// ---- POUs/Components/AxisDriver/Utilities/FB_AxisDistanceTrigger.TcPOU
FUNCTION_BLOCK FB_AxisDistanceTrigger
VAR_INPUT
	/// reset FB
	bReset				: BOOL;
	/// actual position
	fActualPos			: LREAL;
	/// trigger distance
	fTriggerDistance	: LREAL;
END_VAR
VAR_OUTPUT
	/// trigger output
	Q	: BOOL;
END_VAR
VAR PERSISTENT
	/// distance
	fDistance		: LREAL;
	/// actual ABS position
	fActualAbsPos	: LREAL;
	/// mirror ABS position
	fMirrorAbsPos	: LREAL;
	bInit			: BOOL;
END_VAR

fActualAbsPos := ABS(fActualPos);

IF bReset OR NOT bInit THEN
	bInit := TRUE;
	Q := FALSE;
	fMirrorAbsPos := fActualAbsPos;
	IF bReset THEN	
		fDistance := 0;
	END_IF

END_IF

IF fTriggerDistance <= 0 THEN
	Q := FALSE;
	RETURN;
END_IF

IF ABS(fActualAbsPos - fMirrorAbsPos) > fEpsilon THEN
	fDistance := fDistance + ABS(fActualAbsPos - fMirrorAbsPos);
	fMirrorAbsPos := fActualAbsPos;
END_IF

Q := fDistance >= fTriggerDistance;

END_FUNCTION_BLOCK

// ---- POUs/Components/AxisDriver/Utilities/FB_LimitSwitchRefSim.TcPOU
/// Axis driver limit switch
FUNCTION_BLOCK FB_LimitSwitchRefSim
VAR_INPUT
	/// Aktiviert die Logik
	bEnable					:BOOL;
	/// Position der Achse
	fPosition				:REAL;
	
	/// Endschalter (Oeffner)
	bLimitSwitch			:BOOL;
	/// Distanz Simuliertem Ref-Schalter zu Endschalter
	fRefLimitDistance		:REAL := 1.1;
	
	/// Referenzposition
	fRefPosition			:REAL;
	/// Pruefen des Positionsbereichs der Referenzposition
	fRefPosCheckArea		:REAL := 1;
END_VAR
VAR_OUTPUT
	/// Endschalter (Verzeogert)
	bLimitSwitchSim			:BOOL;
	/// Simulierter Ref Schalter
	bRefSwitchSim			:BOOL;
	
	/// Pruefung der Refpos OK
	bRefCheckOk				:BOOL;
END_VAR
VAR
	
END_VAR
VAR PERSISTENT
	fPosLatched			:REAL;
	bPosLatched			:BOOL;
END_VAR

(*
	Baustein um einen Ref-Schalter und Limitswitch mit 1 Eingang zu realisieren
	RE / 2015 / www.rmth.at
*)

// Limit muss hinter Ref liegen
IF (fRefLimitDistance <= fRefPosCheckArea) THEN
	fRefLimitDistance := fRefPosCheckArea + 0.1;
END_IF

IF NOT bEnable THEN
	bLimitSwitchSim := bLimitSwitch;
	bRefSwitchSim := bLimitSwitchSim;
	bRefCheckOk := FALSE;
	RETURN;
END_IF

// logik
IF bLimitSwitch THEN // (oeffner)
	fPosLatched := 0;
	bPosLatched := FALSE;	
	bLimitSwitchSim := TRUE; // limit ok
	bRefSwitchSim := FALSE; // kein referenz
	bRefCheckOk := FALSE;
	
ELSE
	// Position merken
	IF NOT bPosLatched THEN
		bPosLatched := TRUE;
		fPosLatched := fPosition;
	END_IF

	bRefSwitchSim := TRUE;
	bLimitSwitchSim := NOT (ABS(fPosition - fPosLatched) >= fRefLimitDistance);

	// Referenzpunkt pruefen
	bRefCheckOk := (ABS(fRefPosition - fPosLatched) <= fRefPosCheckArea) AND NOT bLimitSwitch;
END_IF

METHOD Reset : bool
VAR_INPUT
END_VAR
fPosLatched := 0;
bPosLatched := FALSE;
END_METHOD

END_FUNCTION_BLOCK

// ---- POUs/Components/AxisDriver/Utilities/F_SpeedReached.TcPOU
/// determines whether the actual speed (ABS value) is within the target-speed window
FUNCTION F_SpeedReached : BOOL
VAR_INPUT
	/// actual speed
	fActualSpeed: LREAL;
	/// target speed
	fTargetSpeed: LREAL;
	/// Override for axis and spindle
	fOverride: LREAL;
END_VAR

F_SpeedReached := F_SpeedWindowReached(fToleranceFactor:=0, fActualSpeed:=fActualSpeed, fTargetSpeed:=fTargetSpeed, fOverride:=fOverride);

END_FUNCTION

// ---- POUs/Components/AxisDriver/Utilities/F_SpeedWindowReached.TcPOU
/// determines whether the actual speed (ABS value) is within the target-speed window
FUNCTION F_SpeedWindowReached : BOOL
VAR_INPUT
	/// factor for tolerance (default: 0.1)
	fToleranceFactor: REAL;
	/// actual speed
	fActualSpeed: LREAL;
	/// target speed
	fTargetSpeed: LREAL;
	/// Override for axis and spindle
	fOverride: LREAL;
END_VAR
VAR CONSTANT
	fDefaultfToleranceFactor: REAL := 0.1;
END_VAR
VAR
	fTol: LREAL;
	fMin: LREAL;
	fMax: LREAL;
	fAct: LREAL;
	fTar: LREAL;
END_VAR

// validate tolerance factor
IF fToleranceFactor <= 0 THEN
	fToleranceFactor:=fDefaultfToleranceFactor;
END_IF

// calc tolerance window and ABS values
fTar:=fTargetSpeed*(fOverride/100);
fTol:=ABS(fTar) * fToleranceFactor;
fMin:=ABS(fTar) - fTol;
fMax:=ABS(fTar) + fTol;
fAct:=ABS(fActualSpeed);

F_SpeedWindowReached := fAct >= fMin AND fAct <= fMax;

END_FUNCTION

// ---- POUs/Components/AxisDriver/Utilities/F_TargetReached.TcPOU
FUNCTION F_TargetReached : BOOL
VAR_INPUT
	fCurrentPos: LREAL;
	fTargetPos: LREAL;
END_VAR

F_TargetReached := F_TargetWindowReached(fCurrentPos, fTargetPos, fEpsilon);

END_FUNCTION

// ---- POUs/Components/AxisDriver/Utilities/F_TargetReachedOrHigher.TcPOU
FUNCTION F_TargetReachedOrHigher : BOOL
VAR_INPUT
	fCurrentPos: LREAL;
	fTargetPos: LREAL;
END_VAR


F_TargetReachedOrHigher := fCurrentPos >= (fTargetPos - fEpsilon);

END_FUNCTION

// ---- POUs/Components/AxisDriver/Utilities/F_TargetReachedOrLower.TcPOU
FUNCTION F_TargetReachedOrLower : BOOL
VAR_INPUT
	fCurrentPos: LREAL;
	fTargetPos: LREAL;
END_VAR


F_TargetReachedOrLower := fCurrentPos <= (fTargetPos + fEpsilon);

END_FUNCTION

// ---- POUs/Components/CylinderDriver/FB_Cylinder_Ui.TcPOU
FUNCTION_BLOCK PUBLIC FB_Cylinder_Ui EXTENDS FB_ManualUiBase
VAR_INPUT
	// Handbetrieb nach GRST
	bManual_HP				: BOOL;
	/// Handbetrieb nach AST
	bManual_WP				: BOOL;
	// Enable Mp
	bEnable_Mp				: BOOL;
END_VAR
VAR_IN_OUT
	// cylinder reference
	fbCylinder				: FB_CylinderEx;
	// hmi control IN
	stHMIControlIn			: ST_HMI_MANUAL_CYLINDER_IN;
	// hmi control IN
	stHMIControlOut			: ST_HMI_MANUAL_CYLINDER_OUT;	
END_VAR
VAR_OUTPUT
	diColorSelectedItem: UDINT;
	/// 0=Undefiniert
	/// 1=Fehler
	/// 2=In GRST (eingefahren)
	/// 3=In AST (ausgefahren) 
	iState: INT;
	diColorState	: UDINT;
	sState			: STRING;
	stState			: ST_Text;
END_VAR

stName.wsName := TO_WSTRING(fbCylinder.sName);
fbCylinder.diObjectIndex := diObjectIndex;
fbCylinder.diSelectedObjectIndex := diSelectedObjectIndex;
fbCylinder.bEnableManual := bEnableManual;
fbCylinder.bManual_HP := stHMIControlIn.stButtonHp.bClick OR ((diObjectIndex = diSelectedObjectIndex) AND stHMIControlIn.stButtonHp.bClick) ;
fbCylinder.bManual_WP := stHMIControlIn.stButtonWp.bClick OR ((diObjectIndex = diSelectedObjectIndex) AND stHMIControlIn.stButtonWp.bClick);

IF ((diObjectIndex = diSelectedObjectIndex) AND stHMIControlIn.stButtonMp.bClick) AND ((fbCylinder.eValveType = E_ValveType.eValvetype_5_3_lock) OR (fbCylinder.eValveType = E_ValveType.eValvetype_5_3_unlock)) THEN
	fbCylinder.ClearOuts();
END_IF

IF (diObjectIndex = diSelectedObjectIndex)AND (diObjectIndex <> 0) AND bEnableManual  THEN
	bManualActive := TRUE;
	stHMIControlOut.bVisible := TRUE;
	stHMIControlOut.stButtonHp.stName := CONST.stTextListGlobal.stText_Hp;
	stHMIControlOut.stButtonMp.stName := CONST.stTextListGlobal.stText_Mp;
	stHMIControlOut.stButtonWp.stName := CONST.stTextListGlobal.stText_Wp;
	stHMIControlOut.stObjectName.wsName := stHMIControlOut.stObjectName.wsNameId := TO_WSTRING(fbCylinder.sName);
	stHMIControlOut.stButtonHp.stColor.color := F_ColorToStringHexColor(STATICS.stColor.Theme);
	stHMIControlOut.stButtonWp.stColor.color := F_ColorToStringHexColor(STATICS.stColor.Theme);
	stHMIControlOut.bMpVisible := bEnable_Mp;
	stHMIControlOut.stButtonMp.stColor.color := F_ColorToStringHexColor(STATICS.stColor.Theme);	
	
	IF fbCylinder.bIn_HP THEN
		stHMIControlOut.stButtonHp.stColor.color := F_ColorToStringHexColor(STATICS.stColor.LimeGreen);
	ELSIF fbCylinder.bIn_WP THEN
		stHMIControlOut.stButtonWp.stColor.color := F_ColorToStringHexColor(STATICS.stColor.LimeGreen);
	END_IF
ELSIF bManualActive THEN
	bManualActive := FALSE;
	stHMIControlOut.bVisible := FALSE;
END_IF

iState := fbCylinder.iStatus;

CASE iState OF 
	1:
		sState:=fbCylinder.sErrText;
		diColorState:= STATICS.stColor.Red;
		stState.wsName := "error";
		stState.wsNameId := "error";
		stState.nNameId := 1;
	2:
		sState:= F_GetTranslatedTxtLib('Zylinder in HP', eLanguage);
		diColorState:= STATICS.stColor.Green;
		stState.wsName := "hp";
		stState.wsNameId := "inhomepos";
		stState.nNameId := 2;		
	3:
		sState:=F_GetTranslatedTxtLib('Zylinder in WP', eLanguage);
		diColorState:= STATICS.stColor.Green;
		stState.wsName := "wp";
		stState.wsNameId := "wp";
		stState.nNameId := 3;
ELSE
	sState:=F_GetTranslatedTxtLib(' Undefiniert ' , eLanguage);	
	diColorState:= STATICS.stColor.Orange;
	stState.wsName := "undifined";
	stState.wsNameId := "undifined";
	stState.nNameId := 0;	
END_CASE


IF (diObjectIndex=diSelectedObjectIndex) THEN
	diColorSelectedItem:=STATICS.stColor.LimeGreen;
ELSE
	diColorSelectedItem:=STATICS.stColor.Gray;	
END_IF

A_StateMapping();

ACTION A_StateMapping:
IF NOT __ISVALIDREF(stStateObject) THEN
	RETURN;
END_IF

// state mapping
stStateObject.stState := stState;
stStateObject.nIndexColor := diColorSelectedItem;
//stStateObject.stValue.wsName := "HP/WP";
END_ACTION

METHOD Control_Hp : BOOL
IF bEnableManual THEN
	bManual_HP:=TRUE;
END_IF
END_METHOD

METHOD Control_Wp : BOOL
IF bEnableManual THEN
	bManual_WP:=TRUE;
END_IF
END_METHOD

END_FUNCTION_BLOCK

// ---- POUs/Components/DriveFu/FB_Drive.TcPOU
FUNCTION_BLOCK FB_Drive
VAR_IN_OUT
	bInHome: BOOL;
END_VAR
VAR_INPUT
	/// component active flag
	bActive: BOOL;
	/// Objekt Name (BMK)
	stName				:ST_Text;
	/// Sicherheit = Freigabe von Bewegungen
	bSafetyOk			:BOOL;
	/// Motorschutz OK
	bMotorprotectionOk		:BOOL;

	// Hand
	///Objekt Index
	diObjectIndex: DINT;
	///Ausgewähltes Objekt in der Visu
	diSelectedObjectIndex	:DINT;
	/// Gibt den Handbetrieb frei
	bEnableManual: BOOL;
	// Handbetrieb nach GRST
	bManual_Reverse: BOOL;
	/// Handbetrieb nach AST
	bManual_Forward: BOOL;
	///	 Handbetrieb Stop
	bManual_Stop :BOOL;
	//	Type Handbetrieb
	// 1 = Tippen
	// 2 = Speichern
	iType : INT;
	
	///	Zus. Freigabe für HP Ausgang schalten	
	bFreigabe_Reverse: BOOL := TRUE;
	///	Zus. Freigabe für WP Ausgang schalten	
	bFreigabe_Forward: BOOL := TRUE;
END_VAR
VAR_OUTPUT	
	/// Summenfehler
	bError		:BOOL;
	/// Fehlerinformation
	sErrText	:ST_Text;
	/// 0=Undefiniert
	/// 1=Fehler
	/// 2=Stillstand OK
	/// 3=Vorwärts
	///	4=Rückwärts 
	iStatus: INT;	

	bInit_OK: BOOL;
	
	bDrive_Reverse_Out: BOOL;
	bDrive_Forward_Out: BOOL;
END_VAR
VAR
	iTypeOld : INT;
	tofForward: TOF;
	tofReverse: TOF;
	
	bDrive_Reverse: BOOL;
	bDrive_Forward: BOOL;
END_VAR

(*FB Drive für Antriebe*)
(*Erstellt von Stephan Schöchtner RMTH GmbH*)
(*21.März.2018*)

tofForward();
tofForward.IN := bManual_Forward;

tofReverse();
tofReverse.IN := bManual_Reverse;


// Initialisierung
IF NOT bInit_OK THEN
	M_Init();	
	bInit_OK :=TRUE;
END_IF

sERRText := CONST.stTextListGlobal.stText_notext;

//Fehler
bError := FALSE;
IF NOT bMotorprotectionOK THEN
	bError := TRUE;
	sErrText := F_CreateDynText("Motorschutz", 0);
END_IF

// Bei Typumschaltung im laufenden Betrieb STOP
IF iType <> iTypeOld THEN
	iTypeOld := iType;
	M_Stop();
END_IF

IF (diObjectIndex = diSelectedObjectIndex) THEN
	// Tippen mit Wendeschützumschaltung und Typumschaltung
	CASE iType OF	//Tippen
	
		1:
			IF bManual_Forward AND NOT bManual_Stop THEN
				bDrive_Reverse := FALSE;
				IF NOT tofReverse.Q THEN
					M_Start_Forward();
				END_IF
			ELSIF bManual_Reverse AND NOT bManual_Stop THEN
				bDrive_Forward := FALSE;
				IF NOT tofForward.Q THEN
					M_Start_Reverse();
				END_IF
			ELSE
				M_Stop();
				//M_Start_Forward := FALSE;
				//M_Start_Reverse := FALSE;
			END_IF
		2:						//Speichern
			IF bManual_Forward AND NOT bManual_Stop THEN
				bDrive_Reverse := FALSE;
				IF NOT tofReverse.Q THEN
					M_Start_Forward();
				END_IF
			ELSIF bManual_Reverse AND NOT bManual_Stop THEN
				bDrive_Forward := FALSE;
				IF NOT tofForward.Q THEN
					M_Start_Reverse();
				END_IF
			END_IF
			IF bManual_Stop THEN
				M_Stop();
				//M_Start_Forward := FALSE;
				//M_Start_Reverse := FALSE;
			END_IF	
	ELSE
		//no type selected
		bError := TRUE;
		sErrText := F_CreateDynText("Handbetriebstyp falsch", 0);
		M_Stop();
	END_CASE
END_IF

IF bError THEN
	istatus := 1;
ELSIF NOT bDrive_Forward AND NOT bDrive_Reverse THEN
	iStatus := 2;
ELSIF bDrive_Forward THEN
	iStatus := 3;
ELSIF bDrive_Reverse THEN
	iStatus := 4;
END_IF


bDrive_Reverse_Out:= bDrive_Reverse AND bFreigabe_Reverse AND bSafetyOk AND bMotorprotectionOk;
bDrive_Forward_Out:= bDrive_Forward AND bFreigabe_Forward AND bSafetyOk AND bMotorprotectionOk;

IF NOT bSafetyOk THEN
	bDrive_Reverse:=FALSE;
	bDrive_Reverse_Out:=FALSE;

	bDrive_Forward:=FALSE;
	bDrive_Forward_Out:=FALSE;	
END_IF


//Wegfahrsperre
IF bError THEN
	M_Stop();
END_IF

METHOD M_Init : BOOL
VAR_INPUT
END_VAR
bDrive_Forward := FALSE;
bDrive_Reverse := FALSE;
tofForward.IN := FALSE;
tofForward.PT := T#150MS;
tofReverse.IN := FALSE;
tofReverse.PT := T#150MS;
END_METHOD

METHOD M_Reset : BOOL
VAR_INPUT
END_VAR
END_METHOD

METHOD M_Start_Forward : BOOL
VAR_INPUT
END_VAR
bDrive_Reverse := FALSE;
bDrive_Forward := TRUE;
END_METHOD

METHOD M_Start_Reverse : BOOL
VAR_INPUT
END_VAR
bDrive_Reverse := TRUE;
bDrive_Forward := FALSE;
END_METHOD

METHOD M_Stop : BOOL
VAR_INPUT
END_VAR
	bDrive_Reverse := FALSE;
	bDrive_Forward := FALSE;
END_METHOD

END_FUNCTION_BLOCK

// ---- POUs/Components/DriveFu/FB_Drive_Ui.TcPOU
FUNCTION_BLOCK PUBLIC FB_Drive_Ui EXTENDS FB_ManualUiBase
VAR_INPUT
	// Handbetrieb Rückwärts
	bManual_Reverse				: BOOL;
	/// Handbetrieb Vorwärts
	bManual_Forward				: BOOL;
	//	Stop
	bManual_Stop				: BOOL;
	//	Type Handmodus
		// 1 = Tippen
		// 2 = Speichern
	iType						: INT;
END_VAR
VAR_IN_OUT
	// drive reference
	fbDrive				: FB_Drive;
	// hmi control IN
	stHMIControlIn			: ST_HMI_MANUAL_DRIVE_IN;
	// hmi control OUT
	stHMIControlOut			: ST_HMI_MANUAL_DRIVE_OUT;	
END_VAR
VAR_OUTPUT
	diColorSelectedItem: UDINT;
	/// 0=Undefiniert
	/// 1=Fehler
	iState: INT;
	diColorState	: UDINT;
	sState			: STRING;
	stState			: ST_Text;
END_VAR

stName := fbDrive.stName;

fbDrive.diObjectIndex := diObjectIndex;
fbDrive.diSelectedObjectIndex := diSelectedObjectIndex;
fbDrive.bEnableManual := bEnableManual;
//fbDrive.bManual_Reverse := bManual_Reverse;
//fbDrive.bManual_Forward := bManual_Forward;
//fbDrive.bManual_Stop := bManual_Stop;
fbDrive.iType := iType;

IF (diSelectedObjectIndex = diObjectIndex)AND (diObjectIndex <> 0) AND bEnableManual THEN
	bManualActive := TRUE;
	stHMIControlOut.bVisible := TRUE;
	stHMIControlOut.stObjectName := fbDrive.stName;
	stHMIControlOut.stButtonJogPos.stName := CONST.stTextListGlobal.stText_Positive;
	stHMIControlOut.stButtonJogNeg.stName := CONST.stTextListGlobal.stText_Negative;
	stHMIControlOut.stButtonStop.stName := CONST.stTextListGlobal.stText_Stop;
	stHMIControlOut.aDriveModeName[0] :=  CONST.stTextListGlobal.stText_Mode_StartStop;
	stHMIControlOut.aDriveModeName[1] :=  CONST.stTextListGlobal.stText_Mode_Jog;
	
	CASE stHMIControlIn.eJogMode OF
		
	E_Drive_JogMode.eJogMode_0 :
			IF stHMIControlIn.stButtonStop.bClick THEN
				fbDrive.M_Stop();
			ELSIF stHMIControlIn.stButtonJogPos.bClick THEN
				fbDrive.M_Start_Forward();
			ELSIF stHMIControlIn.stButtonJogNeg.bClick THEN	
				fbDrive.M_Start_Reverse();	
			END_IF
	E_Drive_JogMode.eJogMode_1 :
		IF stHMIControlIn.stButtonJogPos.bClick THEN
			fbDrive.M_Start_Forward();
		ELSIF stHMIControlIn.stButtonJogNeg.bClick THEN	
			fbDrive.M_Start_Reverse();	
		ELSE
			fbDrive.M_Stop();	
		END_IF				
	END_CASE
	stHMIControlOut.stButtonJogPos.stColor.color := F_ColorToStringHexColor(STATICS.stColor.Theme);
	stHMIControlOut.stButtonJogNeg.stColor.color := F_ColorToStringHexColor(STATICS.stColor.Theme);
	stHMIControlOut.stButtonStop.stColor.color := F_ColorToStringHexColor(STATICS.stColor.Red);
	IF fbDrive.bDrive_Forward_Out THEN
		stHMIControlOut.stButtonJogPos.stColor.color := F_ColorToStringHexColor(STATICS.stColor.LimeGreen);	
	END_IF
	IF fbDrive.bDrive_Reverse_Out THEN
		stHMIControlOut.stButtonJogNeg.stColor.color := F_ColorToStringHexColor(STATICS.stColor.LimeGreen);	
	END_IF	
	
	stHMIControlOut.stState	:= stState;	
ELSIF bManualActive THEN
	bManualActive := FALSE;
	stHMIControlOut.bVisible := FALSE;
END_IF

iState := fbDrive.iStatus;

CASE iState OF 
	1:
		sState:= TO_STRING( fbDrive.sErrText.wsName );
		diColorState:= STATICS.stColor.Red;
		stState.wsName := "error";
		stState.wsNameId := "error";
		stState.nNameId := 1;
	2:
		sState:= ('Stillstand OK');
		diColorState:= STATICS.stColor.Gray;
		stState.wsName := "notmoveing";
		stState.wsNameId := "notmoveing";
		stState.nNameId := 2;
	3:
		sState:= ('Betrieb Vorwärts');
		diColorState:= STATICS.stColor.Green;
		stState.wsName := "movepositive";
		stState.wsNameId := "movepositive";
		stState.nNameId := 3;
	4:
		sState:= ('Betrieb Rückwärts');
		diColorState:= STATICS.stColor.Green;
		stState.wsName := "movenegative";
		stState.wsNameId := "movenegative";
		stState.nNameId := 4;		
				
ELSE
	sState:= (' Undefiniert ');	
	diColorState:= STATICS.stColor.Orange;	
	stState.wsName := "undifined";
	stState.wsNameId := "undifined";
	stState.nNameId := 0;
END_CASE


IF (diObjectIndex=diSelectedObjectIndex) THEN
	diColorSelectedItem:=STATICS.stColor.LimeGreen;
ELSE
	diColorSelectedItem:=STATICS.stColor.Gray;	
END_IF

A_StateMapping();

ACTION A_StateMapping:
IF NOT __ISVALIDREF(stStateObject) THEN
	RETURN;
END_IF

// state mapping
stStateObject.stState := stState;
stStateObject.nIndexColor := diColorSelectedItem;
//stStateObject.stValue.wsName := "mov/stp";
END_ACTION

METHOD Control_Start_Forward : BOOL
IF bEnableManual THEN
	fbDrive.bManual_Reverse := FALSE;
	fbDrive.bManual_Forward := TRUE;
	fbDrive.bManual_Stop := FALSE;	
END_IF
END_METHOD

METHOD Control_Start_Reverse : BOOL
IF bEnableManual THEN
	fbDrive.bManual_Reverse := TRUE;
	fbDrive.bManual_Forward := FALSE;
	fbDrive.bManual_Stop := FALSE;	
END_IF
END_METHOD

METHOD Control_Stop : BOOL
IF bEnableManual THEN
	fbDrive.bManual_Reverse := FALSE;
	fbDrive.bManual_Forward := FALSE;
	fbDrive.bManual_Stop := TRUE;	
END_If
END_METHOD

END_FUNCTION_BLOCK

// ---- POUs/Components/DriveFu/FB_DriveFuAx_Ui.TcPOU
FUNCTION_BLOCK PUBLIC FB_DriveFuAx_Ui EXTENDS FB_ManualUiBase
VAR_INPUT
	// velocity
	fVelocity				: REAL := 1;	
	// additional enable flag for pos. direction
	bEnablePos				: BOOL := TRUE;
	// additional enable flag for neg. direction
	bEnableNeg				: BOOL := TRUE;	
	// manual jog neg.
	bJobN					: BOOL;
	// manual jog pos.
	bJogP					: BOOL;
	// manual stop
	bStop					: BOOL;
END_VAR
VAR_IN_OUT
	// axis reference
	fbAxis				: FB_AxisDriver;
	// hmi control IN
	stHMIControlIn		: ST_HMI_MANUAL_DRIVE_IN;
	// hmi control OUT
	stHMIControlOut		: ST_HMI_MANUAL_DRIVE_OUT;
END_VAR
VAR_OUTPUT	
	diColorSelectedItem: UDINT;
	/// 0=undefined 
	/// 1=error
	/// 2=moving pos. 
	/// 3=moving neg.
	/// 4=standstill
	/// 5=in sync
	iState			: INT;
	diColorState	: UDINT;
	sState			: STRING;
	stState			: ST_Text;
END_VAR
VAR
	stAxisState		: Tc2_MC2.ST_AxisStatus;
END_VAR

// AX5000 UI like frequency inverter (FU)

stName := fbAxis.Name;

// inactive -> reset & exit
IF NOT fbAxis.Active THEN
	stState := CONST.stTextListGlobal.stText_notext;
	iState := 0;// 0=undefined
	A_StateMapping();
	RETURN;
END_IF

IF (diSelectedObjectIndex = diObjectIndex)AND (diObjectIndex <> 0) AND bEnableManual THEN
	bManualActive := TRUE;
	stHMIControlOut.bVisible := TRUE;
	stHMIControlOut.stObjectName := fbAxis.Name;
	stHMIControlOut.stButtonJogPos.stName := CONST.stTextListGlobal.stText_Positive;
	stHMIControlOut.stButtonJogNeg.stName := CONST.stTextListGlobal.stText_Negative;
	stHMIControlOut.stButtonStop.stName := CONST.stTextListGlobal.stText_Stop;
	stHMIControlOut.aDriveModeName[0] :=  CONST.stTextListGlobal.stText_Mode_StartStop;
	stHMIControlOut.aDriveModeName[1] :=  CONST.stTextListGlobal.stText_Mode_Jog;
	
	CASE stHMIControlIn.eJogMode OF
		
	E_Drive_JogMode.eJogMode_0 :
			IF stHMIControlIn.stButtonStop.bClick THEN
				fbAxis.Stop();
			ELSIF stHMIControlIn.stButtonJogPos.bClick THEN
				fbAxis.MoveVel(fVelocity, MC_Direction.MC_Positive_Direction);
			ELSIF stHMIControlIn.stButtonJogNeg.bClick THEN	
				fbAxis.MoveVel(fVelocity, MC_Direction.MC_Negative_Direction);	
			END_IF
	E_Drive_JogMode.eJogMode_1 :
		fbAxis.JogExVel(((bJobN OR stHMIControlIn.stButtonJogNeg.bClick) AND bEnableNeg),
						((bJogP OR stHMIControlIn.stButtonJogPos.bClick) AND bEnablePos),
						fVelocity, E_JogMode.MC_JOGMODE_CONTINOUS);			
	END_CASE
	stHMIControlOut.stButtonJogPos.stColor.color := F_ColorToStringHexColor(STATICS.stColor.Theme);
	stHMIControlOut.stButtonJogNeg.stColor.color := F_ColorToStringHexColor(STATICS.stColor.Theme);
	stHMIControlOut.stButtonStop.stColor.color := F_ColorToStringHexColor(STATICS.stColor.Red);
	IF iState = 2 THEN // 2 = moving neg
		stHMIControlOut.stButtonJogPos.stColor.color := F_ColorToStringHexColor(STATICS.stColor.LimeGreen);	
	END_IF
	IF iState = 3 THEN // 3 = moving neg
		stHMIControlOut.stButtonJogNeg.stColor.color := F_ColorToStringHexColor(STATICS.stColor.LimeGreen);	
	END_IF	
	
	stHMIControlOut.stState	:= stState;	
ELSIF bManualActive THEN
	bManualActive := FALSE;
	stHMIControlOut.bVisible := FALSE;
END_IF

A_StateMapping();

ACTION A_StateMapping:
IF (diObjectIndex = diSelectedObjectIndex) THEN
	diColorSelectedItem := STATICS.stColor.LimeGreen;
ELSE
	diColorSelectedItem := STATICS.stColor.Gray;	
END_IF

bError := fbAxis.State = E_ComponentState.eComponentState_error;
IF bError THEN
	stErrorText := F_CreateDynText(fbAxis.ClearText, 0);
ELSE
	stErrorText := CONST.stTextListGlobal.stText_notext;
END_IF

// Status
stAxisState := fbAxis.AxisState;
IF bError THEN
	iState := 1; // 1=Fehler; 
	diColorState:= STATICS.stColor.Red;
	stState.wsNameId := "error";
	stState.wsName := "error";
	stState.nNameId :=1;
ELSIF stAxisState.Moving AND stAxisState.PositiveDirection THEN
	iState := 2; // 2=Fahrt Positiv; 
	diColorState:= STATICS.stColor.Green;
	stState.wsNameId := "movepositive";
	stState.wsName := "movepositive";
	stState.nNameId :=2;
ELSIF stAxisState.Moving AND stAxisState.NegativeDirection THEN
	iState := 3; // 3=Fahrt Negativ;
	diColorState:= STATICS.stColor.Green;
	stState.wsNameId := "movenegative";
	stState.wsName := "movenegative";
	stState.nNameId :=3;
ELSIF stAxisState.Coupled THEN
	iState := 5; // 5=Synchron
	diColorState:= STATICS.stColor.LightSkyBlue;
	stState.wsNameId := "coupled";
	stState.wsName := "coupled";
	stState.nNameId :=5;
ELSIF NOT stAxisState.Moving THEN
	iState := 4; // 4=Stillstand
	diColorState:= STATICS.stColor.Gray;
	stState.wsNameId := "notmoveing";
	stState.wsName := "notmoveing";
	stState.nNameId :=4;
ELSE
	iState := 0;// 0=Undefiniert
	diColorState:= STATICS.stColor.Orange;
	stState.wsNameId := "undifined";
	stState.wsName := "undifined";
	stState.nNameId :=0;
END_IF

IF NOT __ISVALIDREF(stStateObject) THEN
	RETURN;
END_IF

// state mapping
stStateObject.stState := stState;
stStateObject.nIndexColor := diColorSelectedItem;
//stStateObject.stValue.wsName := "mov/stp";
END_ACTION

END_FUNCTION_BLOCK

// ---- POUs/HMI/Utilities/F_AlarmPrioToText.TcPOU
FUNCTION F_AlarmPrioToText : ST_Text
VAR_INPUT
	ePriority : E_AlarmPriority;
END_VAR

			
CASE ePriority OF
	E_AlarmPriority.Error:
		F_AlarmPrioToText := Const.stTextListGlobal.stText_Error;
		
	E_AlarmPriority.Warning:
		F_AlarmPrioToText := Const.stTextListGlobal.stText_Warning;
		
	ELSE
		F_AlarmPrioToText := Const.stTextListGlobal.stText_Info;
	
END_CASE

END_FUNCTION

// ---- POUs/HMI/Utilities/F_AlarmPrioToHexColor.TcPOU
FUNCTION F_AlarmPrioToHexColor : STRING
VAR_INPUT
	ePriority : E_AlarmPriority;
END_VAR

			
CASE ePriority OF
	E_AlarmPriority.Error:
		F_AlarmPrioToHexColor := F_ColorToStringHexColor(STATICS.stColor.Red);
		
	E_AlarmPriority.Warning:
		F_AlarmPrioToHexColor := F_ColorToStringHexColor(STATICS.stColor.Orange);
		
	ELSE
		F_AlarmPrioToHexColor := F_ColorToStringHexColor(STATICS.stColor.Blue); //F_ColorToStringHexColor(stCol.Theme);
	
END_CASE

END_FUNCTION

// ---- POUs/HMI/Utilities/SettingsHandling/F_SettingItemHandling.TcPOU
FUNCTION F_SettingItemHandling : BOOL
VAR_IN_OUT
	bValue 	: BOOL;
	nValue 	: INT;
	fValue 	: LREAL;
	wsValue	: WSTRING;
	stSetting 	: ST_Data_Item;
END_VAR
VAR
	stInfo 		: ST_Text;
	sChanges	: T_MaxString;
	IEvent		: I_EventHandler;
END_VAR

IF Services.bSettingsSaved OR NOT Services.bPlcInitDone THEN
	bValue := stSetting.bValue;
	nValue := stSetting.nValue;
	fValue := stSetting.fValue;
	wsValue := stSetting.sValue;
	RETURN;
END_IF

IF bValue = stSetting.bValue AND_THEN wsValue = stSetting.sValue AND_THEN
   nValue = stSetting.nValue AND_THEN ABS(fValue - stSetting.fValue) < Statics.fEpsilon THEN
	RETURN;
END_IF

sChanges := sEmpty;
IEvent := Services.fbEventHandler;

// 1. chk user level
IF NOT F_ChkSettingUserLevel(HMI.eUserLevel, stSetting, stInfo => stInfo) THEN
	IEvent.Select(TC_Events.SettingsEventClass.WarningEvent)
		  .ArgAddWString(stInfo.wsName)
		  .Raise();
	
	bValue := stSetting.bValue;
	nValue := stSetting.nValue;
	fValue := stSetting.fValue;
	wsValue := stSetting.sValue;
	RETURN;
END_IF


// 2. chk min/max value
IF NOT F_ChkSettingLimit(nValue, fValue, stSetting, stInfo => stInfo) THEN
	IEvent.Select(TC_Events.SettingsEventClass.WarningEvent)
		  .ArgAddWString(stInfo.wsName)
		  .Raise();
							
	bValue := stSetting.bValue;
	nValue := stSetting.nValue;
	fValue := stSetting.fValue;
	wsValue := stSetting.sValue;
	RETURN;
END_IF

// 3. save changes
IF stSetting.eDataType = E_DataType.eDataType_bool THEN
	F_TrackSettingChangesB(bValue, stSetting, sChanges);
ELSIF stSetting.eDataType = E_DataType.eDataType_int THEN
	F_TrackSettingChangesI(nValue, stSetting, sChanges);
ELSIF stSetting.eDataType = E_DataType.eDataType_lreal THEN
	F_TrackSettingChangesF(fValue, stSetting, sChanges);
ELSIF stSetting.eDataType = E_DataType.eDataType_wstring THEN
	F_TrackSettingChangesWs(wsValue, stSetting, sChanges);
ELSIF stSetting.eDataType = E_DataType.eDataType_time_ms THEN
	F_TrackSettingChangesT(TO_TIME(nValue), stSetting, sChanges);
ELSIF stSetting.eDataType = E_DataType.eDataType_time_s THEN
	F_TrackSettingChangesT(TO_TIME(fValue * 1000), stSetting, sChanges);
ELSIF stSetting.eDataType = E_DataType.eDataType_time_m THEN
	F_TrackSettingChangesT(TO_TIME(fValue * 60000), stSetting, sChanges);
ELSIF stSetting.eDataType = E_DataType.eDataType_time_h THEN
	F_TrackSettingChangesT(TO_TIME(fValue * 360000),stSetting, sChanges);
END_IF

// 4. track settings changes
IF sChanges <> sEmpty THEN
	ILog.AddLog(Concat5('Settings Changed, ', 'EKS level: ', TO_STRING(HMI.eUserLevel), '. Changes: ', sChanges), 
				'HMI Controller', 
				E_LogLevel.eLogLevel_info);
END_IF

bValue := stSetting.bValue;
nValue := stSetting.nValue;
fValue := stSetting.fValue;
wsValue := stSetting.sValue;

END_FUNCTION

// ---- POUs/HMI/Utilities/SettingsHandling/F_SettingItemHandlingB.TcPOU
FUNCTION F_SettingItemHandlingB : BOOL
VAR_IN_OUT
	bValue 		: BOOL;
	stSetting 	: ST_Data_Item;
END_VAR
VAR
	stInfo 		: ST_Text;
	sChanges	: T_MaxString;
	IEvent		: I_EventHandler;
END_VAR

F_SettingItemHandlingB := stSetting.bValue;

IF Services.bSettingsSaved OR NOT Services.bPlcInitDone THEN
	bValue := stSetting.bValue;
	RETURN;
END_IF

IF bValue = stSetting.bValue THEN
	RETURN;
END_IF

sChanges := sEmpty;
IEvent := Services.fbEventHandler;

// 1. chk user level
IF NOT F_ChkSettingUserLevel(HMI.eUserLevel, stSetting, stInfo => stInfo) THEN							  
	IEvent.Select(TC_Events.SettingsEventClass.WarningEvent)
		  .ArgAddWString(stInfo.wsName)
		  .Raise();
							
	bValue := stSetting.bValue;
	RETURN;
END_IF


// 2. chk min/max value
//IF NOT F_ChkSettingLimit(nValue, fValue, stSetting, stInfo => stInfo) THEN
//	IEvent.Select(TC_Events.SettingsEventClass.WarningEvent)
//		  .ArgAddWString(stInfo.wsName)
//		  .Raise();
//							
//	bValue := stSetting.bValue;
//	RETURN;
//END_IF

// 3. save changes
IF stSetting.eDataType = E_DataType.eDataType_bool THEN
	F_TrackSettingChangesB(bValue, stSetting, sChanges);
ELSIF stSetting.eDataType = E_DataType.eDataType_int THEN
	F_TrackSettingChangesI(TO_INT(bValue), stSetting, sChanges);
ELSIF stSetting.eDataType = E_DataType.eDataType_lreal THEN
	F_TrackSettingChangesF(TO_LREAL(bValue), stSetting, sChanges);
ELSIF stSetting.eDataType = E_DataType.eDataType_wstring THEN
	F_TrackSettingChangesWs(TO_WSTRING(bValue), stSetting, sChanges);
ELSIF stSetting.eDataType = E_DataType.eDataType_time_ms THEN
	F_TrackSettingChangesT(TO_TIME(bValue), stSetting, sChanges);
ELSIF stSetting.eDataType = E_DataType.eDataType_time_s THEN
	F_TrackSettingChangesT(TO_TIME(TO_INT(bValue) * 1000), stSetting, sChanges);
ELSIF stSetting.eDataType = E_DataType.eDataType_time_m THEN
	F_TrackSettingChangesT(TO_TIME(TO_INT(bValue) * 60000), stSetting, sChanges);
ELSIF stSetting.eDataType = E_DataType.eDataType_time_h THEN
	F_TrackSettingChangesT(TO_TIME(TO_INT(bValue) * 360000),stSetting, sChanges);
END_IF

// 4. track settings changes
IF sChanges <> sEmpty THEN
	ILog.AddLog(Concat5('Settings Changed, ', 'EKS level: ', TO_STRING(HMI.eUserLevel), '. Changes: ', sChanges), 
				'HMI Controller', 
				E_LogLevel.eLogLevel_info);
END_IF

bValue := stSetting.bValue;
F_SettingItemHandlingB := stSetting.bValue;

END_FUNCTION

// ---- POUs/HMI/Utilities/SettingsHandling/F_SettingItemHandlingF.TcPOU
FUNCTION F_SettingItemHandlingF : LREAL
VAR_IN_OUT
	fValue 		: LREAL;
	stSetting 	: ST_Data_Item;
END_VAR
VAR
	stInfo 		: ST_Text;
	sChanges	: T_MaxString;
	IEvent		: I_EventHandler;
END_VAR

F_SettingItemHandlingF := stSetting.fValue;

IF Services.bSettingsSaved OR NOT Services.bPlcInitDone THEN
	fValue := stSetting.fValue;
	RETURN;
END_IF

IF ABS(fValue - stSetting.fValue) < Statics.fEpsilon THEN
	RETURN;
END_IF

sChanges := sEmpty;
IEvent := Services.fbEventHandler;

// 1. chk user level
IF NOT F_ChkSettingUserLevel(HMI.eUserLevel, stSetting, stInfo => stInfo) THEN							  
	IEvent.Select(TC_Events.SettingsEventClass.WarningEvent)
		  .ArgAddWString(stInfo.wsName)
		  .Raise();
							
	fValue := stSetting.fValue;
	RETURN;
END_IF


// 2. chk min/max value
IF NOT F_ChkSettingLimitF(fValue, stSetting, stInfo => stInfo) THEN
	IEvent.Select(TC_Events.SettingsEventClass.WarningEvent)
		  .ArgAddWString(stInfo.wsName)
		  .Raise();
							
	fValue := stSetting.fValue;
	RETURN;
END_IF

// 3. save changes
IF stSetting.eDataType = E_DataType.eDataType_bool THEN
	F_TrackSettingChangesB(fValue = 1, stSetting, sChanges);
ELSIF stSetting.eDataType = E_DataType.eDataType_int THEN
	F_TrackSettingChangesI(TO_INT(fValue), stSetting, sChanges);
ELSIF stSetting.eDataType = E_DataType.eDataType_lreal THEN
	F_TrackSettingChangesF(fValue, stSetting, sChanges);
ELSIF stSetting.eDataType = E_DataType.eDataType_wstring THEN
	F_TrackSettingChangesWs(TO_WSTRING(fValue), stSetting, sChanges);
ELSIF stSetting.eDataType = E_DataType.eDataType_time_ms THEN
	F_TrackSettingChangesT(TO_TIME(fValue), stSetting, sChanges);
ELSIF stSetting.eDataType = E_DataType.eDataType_time_s THEN
	F_TrackSettingChangesT(TO_TIME(fValue * 1000), stSetting, sChanges);
ELSIF stSetting.eDataType = E_DataType.eDataType_time_m THEN
	F_TrackSettingChangesT(TO_TIME(fValue * 60000), stSetting, sChanges);
ELSIF stSetting.eDataType = E_DataType.eDataType_time_h THEN
	F_TrackSettingChangesT(TO_TIME(fValue * 360000),stSetting, sChanges);
END_IF

// 4. track settings changes
IF sChanges <> sEmpty THEN
	ILog.AddLog(Concat5('Settings Changed, ', 'EKS level: ', TO_STRING(HMI.eUserLevel), '. Changes: ', sChanges), 
				'HMI Controller', 
				E_LogLevel.eLogLevel_info);
END_IF

fValue := stSetting.fValue;
F_SettingItemHandlingF := stSetting.fValue;

END_FUNCTION

// ---- POUs/HMI/Utilities/SettingsHandling/F_SettingItemHandlingI.TcPOU
FUNCTION F_SettingItemHandlingI : INT
VAR_IN_OUT
	nValue 		: INT;
	stSetting 	: ST_Data_Item;
END_VAR
VAR
	stInfo 		: ST_Text;
	sChanges	: T_MaxString;
	IEvent		: I_EventHandler;
END_VAR

F_SettingItemHandlingI := stSetting.nValue;

IF Services.bSettingsSaved OR NOT Services.bPlcInitDone THEN
	nValue := stSetting.nValue;
	RETURN;
END_IF

IF nValue = stSetting.nValue THEN
	RETURN;
END_IF

sChanges := sEmpty;
IEvent := Services.fbEventHandler;

// 1. chk user level
IF NOT F_ChkSettingUserLevel(HMI.eUserLevel, stSetting, stInfo => stInfo) THEN							  
	IEvent.Select(TC_Events.SettingsEventClass.WarningEvent)
		  .ArgAddWString(stInfo.wsName)
		  .Raise();
							
	nValue := stSetting.nValue;
	RETURN;
END_IF


// 2. chk min/max value
IF NOT F_ChkSettingLimitN(nValue, stSetting, stInfo => stInfo) THEN
	IEvent.Select(TC_Events.SettingsEventClass.WarningEvent)
		  .ArgAddWString(stInfo.wsName)
		  .Raise();
							
	nValue := stSetting.nValue;
	RETURN;
END_IF

// 3. save changes
IF stSetting.eDataType = E_DataType.eDataType_bool THEN
	F_TrackSettingChangesB(nValue = 1, stSetting, sChanges);
ELSIF stSetting.eDataType = E_DataType.eDataType_int THEN
	F_TrackSettingChangesI(TO_INT(nValue), stSetting, sChanges);
ELSIF stSetting.eDataType = E_DataType.eDataType_lreal THEN
	F_TrackSettingChangesF(TO_REAL(nValue), stSetting, sChanges);
ELSIF stSetting.eDataType = E_DataType.eDataType_wstring THEN
	F_TrackSettingChangesWs(TO_WSTRING(nValue), stSetting, sChanges);
ELSIF stSetting.eDataType = E_DataType.eDataType_time_ms THEN
	F_TrackSettingChangesT(TO_TIME(nValue), stSetting, sChanges);
ELSIF stSetting.eDataType = E_DataType.eDataType_time_s THEN
	F_TrackSettingChangesT(TO_TIME(nValue * 1000), stSetting, sChanges);
ELSIF stSetting.eDataType = E_DataType.eDataType_time_m THEN
	F_TrackSettingChangesT(TO_TIME(nValue * 60000), stSetting, sChanges);
ELSIF stSetting.eDataType = E_DataType.eDataType_time_h THEN
	F_TrackSettingChangesT(TO_TIME(nValue * 360000),stSetting, sChanges);
END_IF

// 4. track settings changes
IF sChanges <> sEmpty THEN
	ILog.AddLog(Concat5('Settings Changed, ', 'EKS level: ', TO_STRING(HMI.eUserLevel), '. Changes: ', sChanges), 
				'HMI Controller', 
				E_LogLevel.eLogLevel_info);
END_IF

nValue := stSetting.nValue;
F_SettingItemHandlingI := stSetting.nValue;

END_FUNCTION

// ---- POUs/HMI/Utilities/SettingsHandling/F_SettingItemHandlingWs.TcPOU
FUNCTION F_SettingItemHandlingWs : WSTRING
VAR_IN_OUT
	wsValue		: WSTRING;
	stSetting 	: ST_Data_Item;
END_VAR
VAR
	stInfo 		: ST_Text;
	sChanges	: T_MaxString;
	IEvent		: I_EventHandler;
END_VAR

F_SettingItemHandlingWs := stSetting.sValue;

IF Services.bSettingsSaved OR NOT Services.bPlcInitDone THEN
	wsValue := stSetting.sValue;
	RETURN;
END_IF

IF wsValue = stSetting.sValue THEN
	RETURN;
END_IF

sChanges := sEmpty;
IEvent := Services.fbEventHandler;

// 1. chk user level
IF NOT F_ChkSettingUserLevel(HMI.eUserLevel, stSetting, stInfo => stInfo) THEN							  
	IEvent.Select(TC_Events.SettingsEventClass.WarningEvent)
		  .ArgAddWString(stInfo.wsName)
		  .Raise();
							
	wsValue := stSetting.sValue;
	RETURN;
END_IF


// 2. chk min/max value
//IF NOT F_ChkSettingLimitF(wsValue, stSetting, stInfo => stInfo) THEN
//	IEvent.Select(TC_Events.SettingsEventClass.WarningEvent)
//		  .ArgAddWString(stInfo.wsName)
//		  .Raise();
//							
//	wsValue := stSetting.sValue;
//	RETURN;
//END_IF

// 3. save changes

IF stSetting.eDataType = E_DataType.eDataType_wstring THEN
	F_TrackSettingChangesWs(wsValue, stSetting, sChanges);
END_IF

// 4. track settings changes
IF sChanges <> sEmpty THEN
	ILog.AddLog(Concat5('Settings Changed, ', 'EKS level: ', TO_STRING(HMI.eUserLevel), '. Changes: ', sChanges), 
				'HMI Controller', 
				E_LogLevel.eLogLevel_info);
END_IF

wsValue := stSetting.sValue;
F_SettingItemHandlingWs := stSetting.sValue;

END_FUNCTION

// ---- POUs/Safety/Components/Euchner_MBM/FB_Euchner_MBM.TcPOU
FUNCTION_BLOCK FB_Euchner_MBM
VAR_INPUT
	stHwIn: ST_Euchner_MBM_HW_IN;
	bReset: BOOL;
END_VAR
VAR_OUTPUT
	stHwOut: ST_Euchner_MBM_HW_OUT;
	bError: BOOL;
	stErrorText: ST_Text;
END_VAR
VAR
	stIn: ST_Euchner_MBM_IN;
	stOut: ST_Euchner_MBM_Out;
	tonReset: ton;
END_VAR

M_Mapping();
M_Supervision();

tonReset.IN := bReset;
tonReset.PT := T#150MS;
tonReset();
IF tonReset.Q THEN
	bReset := FALSE;
END_IF
stOut.bBM_ACK_G := bReset;

METHOD PRIVATE M_Error : BOOL
VAR_INPUT
	stError: ST_Text;
END_VAR
bError	:=TRUE;
stErrorText	:= stError;
END_METHOD

METHOD PRIVATE M_Mapping : BOOL
//mapping in
stIn.bBM_D_RUN := stHwIn.nByte0.0;
stIn.bBM_E_ML1 := stHwIn.nByte0.1;
stIn.bBM_E_ML2 := stHwIn.nByte0.2;
stIn.bBM_E_SYS := stHwIn.nByte0.3;
stIn.bBM_E_G := stHwIn.nByte0.4;

//mapping in
stHwOut.nByte0.0 := stOut.bBM_ACK_G;
END_METHOD

METHOD M_Reset : BOOL
bReset	:= TRUE;
bError	:= FALSE;
MEMSET(ADR(stErrorText), 0, SiZEOF(stErrorText));
END_METHOD

METHOD PRIVATE M_Supervision : BOOL
IF stIn.bBM_E_ML1 THEN
	M_Error(F_CreateDynTextDefault("Fehler Modul MBM Starng 1")); 	
ELSIF stIn.bBM_E_ML1 THEN
	M_Error(F_CreateDynTextDefault("Fehler Modul MBM Starng 1"));	
ELSIF stIn.bBM_E_G THEN
	M_Error(F_CreateDynTextDefault("Modul MBM Allgemein"));	
ELSIF stIn.bBM_E_SYS THEN
	M_Error(F_CreateDynTextDefault("Fehler Gesamtsystem"));
END_IF
END_METHOD

END_FUNCTION_BLOCK

// ---- POUs/System/Supervision/ImplicitChecks/CheckBounds.TcPOU
/// Implicitly generated code : DO NOT EDIT!!!
/// CheckBounds is used to check for range overflows
{attribute 'check_bounds' := ''}
{attribute 'no_check' := ''}
FUNCTION CheckBounds : DINT
VAR_INPUT
	index: DINT;
	lower: DINT;
	upper: DINT;
END_VAR

// align bounds 
CheckBounds := MIN(upper, MAX(lower, index));

// if index changed, report error
IF CheckBounds <> index THEN
	Services.fbEventHandler.Select(TC_Events.CodeEventClass.ErrorEvent)
						   .ArgSetString('check bounds')
						   .Raise();
END_IF

END_FUNCTION

// ---- POUs/System/Supervision/ImplicitChecks/CheckDivDInt.TcPOU
/// Implicitly generated code : DO NOT EDIT!!!
/// Checks for division by 0, if divisor is 0, replace it with 1 and report error
{attribute 'check_div_int32' := ''}
{attribute 'no_check' := ''}
FUNCTION CheckDivDInt : DINT
VAR_INPUT
	divisor: DINT;
END_VAR

IF divisor = 0 THEN
	// replace divisor and report error if necessary
	CheckDivDInt := 1;
	Services.fbEventHandler.Select(TC_Events.CodeEventClass.ErrorEvent)
						   .ArgSetString('div 0 DINT')
						   .Raise();
ELSE
	CheckDivDInt := divisor;
END_IF;

END_FUNCTION

// ---- POUs/System/Supervision/ImplicitChecks/CheckDivLInt.TcPOU
/// Implicitly generated code : DO NOT EDIT!!!
/// Checks for division by 0, if divisor is 0, replace it with 1 and report error
{attribute 'no_check' := ''}
{attribute 'check_div_int64' := ''}
FUNCTION CheckDivLInt : LINT
VAR_INPUT
	divisor: LINT;
END_VAR

IF divisor = 0 THEN
	// replace divisor and report error if necessary
	CheckDivLInt := 1;
	Services.fbEventHandler.Select(TC_Events.CodeEventClass.ErrorEvent)
						   .ArgSetString('div 0 LINT')
						   .Raise();
ELSE
	CheckDivLInt := divisor;
END_IF;

END_FUNCTION

// ---- POUs/System/Supervision/ImplicitChecks/CheckDivLReal.TcPOU
/// Implicitly generated code : DO NOT EDIT!!!
/// Checks for division by 0, if divisor is 0, replace it with 1 and report error
{attribute 'no_check' := ''}
{attribute 'check_div_real64' := ''}
FUNCTION CheckDivLReal : LREAL
VAR_INPUT
	divisor: LREAL;
END_VAR

IF divisor = 0 THEN
	// replace divisor and report error if necessary
	CheckDivLReal := 1;
	Services.fbEventHandler.Select(TC_Events.CodeEventClass.ErrorEvent)
						   .ArgSetString('div 0 LREAL')
						   .Raise();
ELSE
	CheckDivLReal:=divisor;
END_IF;

END_FUNCTION

// ---- POUs/System/Supervision/ImplicitChecks/CheckDivReal.TcPOU
/// Implicitly generated code : DO NOT EDIT
/// Checks for division by 0, if divisor is 0, replace it with 1 and report error
{attribute 'check_div_real32' := ''}
{attribute 'no_check' := ''}
FUNCTION CheckDivReal : REAL
VAR_INPUT
	divisor: REAL;
END_VAR

IF divisor = 0 THEN
	// replace divisor and report error if necessary
	CheckDivReal := 1;
	Services.fbEventHandler.Select(TC_Events.CodeEventClass.ErrorEvent)
						   .ArgSetString('div 0 REAL')
						   .Raise();
ELSE
	CheckDivReal := divisor;
END_IF;

END_FUNCTION

// ---- POUs/System/Supervision/ImplicitChecks/CheckPointer.TcPOU
/// Implicitly generated code : DO NOT EDIT!!!
/// checks for correct pointer use. Currently, this only detects null pointer, which are replaced by 
/// a pointer to a dummy area and reported as error
{attribute 'check_pointer' := ''}
{attribute 'no_check' := ''}
FUNCTION CheckPointer : POINTER TO BYTE
VAR_INPUT
	/// Destination address of the pointer
	ptToTest: POINTER TO BYTE;
	/// Size of the type the pointer points to. (e.g: 20 for POINTER TO ARRAY [0..9] OF INT) 
	iSize: DINT;
	/// Granularity of the pointer access. This is the size of the biggest non-structured data type in the type the pointer points to. (e.g: 2 for POINTER TO ARRAY [0..9] OF INT)
	iGran: DINT;
	/// Indicates read or write Access. TRUE = write access.
	bWrite: BOOL;
END_VAR

// check for outside address range
IF ptToTest = 0 THEN
	// report error 
	Services.fbEventHandler.Select(TC_Events.CodeEventClass.ErrorEvent)
						   .ArgSetString('pointer')
						   .Raise();
	// this is just a desparate way to keep the PLC from crashing, 
	// probably there's a better solution
	CheckPointer := ADR( MAIN ); 
END_IF

END_FUNCTION

// ---- POUs/System/Supervision/ImplicitChecks/CheckRangeSigned.TcPOU
/// Implicitly generated code : DO NOT EDIT!!!
/// Checks subrange value. If value is outside [lower,upper], it is set to the closer bound and reports the error.
{attribute 'check_range_signed' := ''}
{attribute 'no_check' := ''}
FUNCTION CheckRangeSigned : DINT
VAR_INPUT
	value: DINT;
	lower: DINT;
	upper: DINT;
END_VAR

// align to bounds 
CheckRangeSigned := MIN( upper, MAX( lower, value ));

// if value changed, report error
IF CheckRangeSigned <> value THEN
	Services.fbEventHandler.Select(TC_Events.CodeEventClass.ErrorEvent)
						   .ArgSetString('range signed')
						   .Raise();
END_IF

END_FUNCTION

// ---- POUs/System/Supervision/ImplicitChecks/CheckRangeUnsigned.TcPOU
/// Implicitly generated code : DO NOT EDIT
/// Checks subrange value. If value is outside [lower,upper], it is set to the closer bound and reports the error.
{attribute 'check_range_unsigned' := ''}
{attribute 'no_check' := ''}
FUNCTION CheckRangeUnsigned : UDINT
VAR_INPUT
	value: UDINT;
	lower: UDINT;
	upper: UDINT;
END_VAR

// align to bounds 
CheckRangeUnsigned := MIN(upper, MAX(lower, value));

// if value changed, report error
IF CheckRangeUnsigned <> value THEN
	Services.fbEventHandler.Select(TC_Events.CodeEventClass.ErrorEvent)
						   .ArgSetString('range unsigned')
						   .Raise();
END_IF

END_FUNCTION

// ---- POUs/System/Utilities/Convert/F_DegPerSecToDegPerMin.TcPOU
FUNCTION F_DegPerSecToDegPerMin : LREAL
VAR_INPUT
	fValue : LREAL; // °/s value
END_VAR
VAR
END_VAR

 F_DegPerSecToDegPerMin := fValue * 60; // °/s -> °/min

END_FUNCTION

// ---- POUs/System/Utilities/Convert/F_DegPerSecToUpm.TcPOU
FUNCTION F_DegPerSecToUpm : LREAL
VAR_INPUT
	fValue : LREAL; // °/s value
END_VAR
VAR
END_VAR

F_DegPerSecToUpm := fValue * 1/6; // °/s => 1/min (x * 60/360)

END_FUNCTION

// ---- POUs/System/Utilities/Convert/F_Diagnostic_EcDeviceState.TcPOU
/// Function convert EtherCat device state from a slave into an text
FUNCTION F_Diagnostic_EcDeviceState : WSTRING(80)
VAR_INPUT
	/// Function input
	nDeviceState			:BYTE;
END_VAR
VAR
END_VAR

CASE nDeviceState OF
	EC_DEVICE_STATE_INIT:
		F_Diagnostic_EcDeviceState := "EtherCat Device State: INIT";
		
	EC_DEVICE_STATE_PREOP:
		F_Diagnostic_EcDeviceState := "EtherCat Device State: Pre-Operational";
		
	EC_DEVICE_STATE_BOOTSTRAP:
		F_Diagnostic_EcDeviceState := "EtherCat Device State: Bootstrap";
		
	EC_DEVICE_STATE_SAFEOP:
		F_Diagnostic_EcDeviceState := "EtherCat Device State: Safe-Operational";
		
	EC_DEVICE_STATE_OP:
		F_Diagnostic_EcDeviceState := "EtherCat Device State: Operational";
		
	EC_DEVICE_STATE_ERROR:
		F_Diagnostic_EcDeviceState := "EtherCat Device State: Statemachine-error in slave";
		
	EC_DEVICE_STATE_INVALID_VPRS:
		F_Diagnostic_EcDeviceState := "EtherCat Device State: Invalid VendorID, Productcode, revisionnumber or serialnumber";
		
	EC_DEVICE_STATE_INITCMD_ERROR:
		F_Diagnostic_EcDeviceState := "EtherCat Device State: INIT command error";
		
	ELSE 
		F_Diagnostic_EcDeviceState := "EtherCat Device State: Undefined";
END_CASE

END_FUNCTION

// ---- POUs/System/Utilities/Convert/F_Diagnostic_EcLinkState.TcPOU
/// Function convert EtherCat link state from a slave into an text
FUNCTION F_Diagnostic_EcLinkState : WSTRING(80)
VAR_INPUT
	/// Function input
	nLinkState				:BYTE;
END_VAR
VAR
END_VAR

CASE nLinkState OF
	EC_LINK_STATE_OK:
		F_Diagnostic_EcLinkState := "EtherCat Link State: OK";
		
	EC_LINK_STATE_NOT_PRESENT:
		F_Diagnostic_EcLinkState := "EtherCat Link State: No EtherCat communication with EtherCat slave";
		
	EC_LINK_STATE_LINK_WITHOUT_COMM:
		F_Diagnostic_EcLinkState := "EtherCat Link State: Error on port X. Port has a link, but no communication";
		
	EC_LINK_STATE_MISSING_LINK:
		F_Diagnostic_EcLinkState := "EtherCat Link State: Missing link on port X";
		
	EC_LINK_STATE_ADDITIONAL_LINK:
		F_Diagnostic_EcLinkState := "EtherCat Link State: Additional link on port X";
		
	EC_LINK_STATE_PORT_A:
		F_Diagnostic_EcLinkState := "EtherCat Link State: Error communication port A";
		
	EC_LINK_STATE_PORT_B:
		F_Diagnostic_EcLinkState := "EtherCat Link State: Error communication port B";
		
	EC_LINK_STATE_PORT_C:
		F_Diagnostic_EcLinkState := "EtherCat Link State: Error communication port C";
		
	EC_LINK_STATE_PORT_D:
		F_Diagnostic_EcLinkState := "EtherCat Link State: Error communication port D";
		
	ELSE 
		F_Diagnostic_EcLinkState := "EtherCat Link State: Undefined";
END_CASE

END_FUNCTION

// ---- POUs/System/Utilities/Convert/F_Diagnostic_EcMasterDeviceState.TcPOU
/// Function convert EtherCat master device state into an text
FUNCTION F_Diagnostic_EcMasterDeviceState : WSTRING(80)
VAR_INPUT
	/// Function input
	nDeviceState			:UINT;
END_VAR
VAR
END_VAR

CASE nDeviceState OF
	// Link error
	16#1:
		F_Diagnostic_EcMasterDeviceState := "EtherCat: Link error";
		
	// I/O locked after link error (I/O reset required)
	16#2:
		F_Diagnostic_EcMasterDeviceState := "EtherCat: I/O locked after link error (I/O reset required)";
		
	// Link error (redundancy adapter)
	16#4:
		F_Diagnostic_EcMasterDeviceState := "EtherCat: Link error (redundancy adapter)";
		
	// Missing one frame (redundancy mode)
	16#8:
		F_Diagnostic_EcMasterDeviceState := "EtherCat: Missing one frame (redundancy mode)";
		
	// Out of send resources (I/O reset required)
	16#10:
		F_Diagnostic_EcMasterDeviceState := "EtherCat: Out of send resources (I/O reset required)";
		
	// Watchdog triggered
	16#20:
		F_Diagnostic_EcMasterDeviceState := "EtherCat: Watchdog triggered";
		
	// Ethernet driver (miniport) not found
	16#40:
		F_Diagnostic_EcMasterDeviceState := "EtherCat: Ethernet driver (miniport) not found";
		
	// I/O reset active
	16#80:
		F_Diagnostic_EcMasterDeviceState := "EtherCat: I/O reset active";
		
	// At least one device in "INIT" state
	16#100:
		F_Diagnostic_EcMasterDeviceState := "EtherCat: At least one device in INIT state";
		
	// At least one device in "PRE-OP" state
	16#200:
		F_Diagnostic_EcMasterDeviceState := "EtherCat: At least one device in PRE-OP state";
		
	// At least one device in "SAFE-OP" state
	16#400:
		F_Diagnostic_EcMasterDeviceState := "EtherCat: At least one device in SAFE-OP state";
		
	// At least one device indicates an error state
	16#800:
		F_Diagnostic_EcMasterDeviceState := "EtherCat: At least one device indicates an error state";
		
	// DC not in sync
	16#1000:
		F_Diagnostic_EcMasterDeviceState := "EtherCat: DC not in sync";
		
	ELSE 
		F_Diagnostic_EcMasterDeviceState := WCONCAT("EtherCat error: ", UINT_TO_WSTRING(nDeviceState));
END_CASE

END_FUNCTION

// ---- POUs/System/Utilities/Convert/F_MeterPerMinToMmPerSec.TcPOU
FUNCTION F_MeterPerMinToMmPerSec : LREAL
VAR_INPUT
	fValue : LREAL; // m/min value
END_VAR
VAR
END_VAR

 F_MeterPerMinToMmPerSec := fValue * 100/6; // m/min -> mm/s -> x * 1000/60

END_FUNCTION

// ---- POUs/System/Utilities/Convert/F_MmPerSecToMmPerMin.TcPOU
FUNCTION F_MmPerSecToMmPerMin : LREAL
VAR_INPUT
	fValue : LREAL; // mm/s value
END_VAR
VAR
END_VAR

 F_MmPerSecToMmPerMin := fValue * 60; // mm/s -> mm/min -> x * 60

END_FUNCTION

// ---- POUs/System/Utilities/Convert/F_UpmToDegreePerSec.TcPOU
FUNCTION F_UpmToDegreePerSec : LREAL
VAR_INPUT
	fValue : LREAL; // 1/min value
END_VAR
VAR
END_VAR

 F_UpmToDegreePerSec := fValue * 6; // 1/min -> °/s => x * 360/60

END_FUNCTION

// ---- POUs/System/Utilities/Convert/F_MmPerMinToMmPerSec.TcPOU
FUNCTION F_MmPerMinToMmPerSec : LREAL
VAR_INPUT
	fValue : LREAL; // mm/min value
END_VAR
VAR
END_VAR

 F_MmPerMinToMmPerSec := fValue/60; // mm/min -> mm/s -> x * 1/60

END_FUNCTION

// ---- POUs/System/Utilities/Convert/F_MmPerSecToMeterPerMin.TcPOU
FUNCTION F_MmPerSecToMeterPerMin : LREAL
VAR_INPUT
	fValue : LREAL; // mm/s value
END_VAR
VAR
END_VAR

 F_MmPerSecToMeterPerMin := fValue * 6E-2;	// mm/s -> m/min => 60/1000

END_FUNCTION

// ---- POUs/System/Utilities/Convert/F_DegPerMinToDegPerSec.TcPOU
FUNCTION F_DegPerMinToDegPerSec : LREAL
VAR_INPUT
	fValue : LREAL; // °/min value
END_VAR
VAR
END_VAR

 F_DegPerMinToDegPerSec := fValue/60; // °/min -> °/s

END_FUNCTION

// ---- POUs/System/Utilities/CSV/FB_WriteCSV.TcPOU
FUNCTION_BLOCK FB_WriteCSV EXTENDS FB_LoggerBase
VAR_INPUT
	sSource			: STRING := 'PLC';
	sPath			: STRING := 'C:\Temp';
	sYear			: STRING := '2020';
	sMonth			: STRING := '09';
	sDay			: STRING := '28';
	sFileName		: STRING := 'file.csv';
	tWriteFilter	: TIME := T#1M;
END_VAR
VAR_OUTPUT
	/// Fehler
	bError			: BOOL;
	sErrorString	: WSTRING(255);
END_VAR
VAR
	bInit 			: BOOL;
	fbDirectory		: FB_Directory;
	sPath_OLD		: STRING;
	///	log structure		
	//stLog			: REFERENCE TO ST_FileLog;	
	stOrderData		: REFERENCE TO ST_FillOrder;
		
	///	fbs	
	fbFileOpen		: FB_FileOpen;
	fbFileWrite		: FB_FileWrite;
	fbFileClose		: FB_FileClose;
	fbFileRename	: FB_FileRename;
	fbEOF			: FB_EOF;
	fbFindDir		: FB_EnumFindFileEntry;
	sFindDirComp	: STRING;
	
	///	full path
	sFullPath		: STRING;
	sPathNew		: STRING;
	
	// file handle
	hFile			: UINT;
	
	//storaged Message
	saMessage		: ARRAY[0..iMaxIdxCsvData] OF WSTRING(255);
	iMessageCount	: INT;
	sText 			: STRING(255);
	bStartWrite		: BOOL;
	
	///	step flow file logging	
	nStep			: INT;
	tonDelay		: TON;
	
	tonDelayDirectoryExist	:TON;
	
	// log buffer	
	aLogBuffer		: (*ARRAY[0..iMaxIdxLogBuffer] OF*) ST_FillOrder;
	aWriteBuffer	: (*ARRAY[0..iMaxIdxLogBuffer] OF*) ST_FillOrder;
	
END_VAR
VAR CONSTANT
	iMaxIdxCsvData		: INT := 20;
	iMaxIdxLogBuffer	: INT := 1;
END_VAR

THIS^.Run();

METHOD PRIVATE Init : BOOL
VAR_INPUT
END_VAR
Init := bInit;
IF Init THEN
	fbFindDir.bExecute:=FALSE;
	RETURN;
END_IF


fbFindDir(
	sNetId:= , 
	sPathName:=sPath , 
	eCmd:=E_EnumCmdType.eEnumCmd_First , 
	bExecute:=TRUE , 
	tTimeout:= , 
	bBusy=> , 
	bError=> , 
	nErrID=> , 
	bEOE=> , 
	stFindFile=> );
	
	


fbDirectory.Create(sPath);
fbDirectory();

sFindDirComp:=DELETE(sPath,3,1);

bInit := fbDirectory.bDirectoryExist; // OR (fbFindDir.stFindFile.sFileName = sFindDirComp);

IF NOT bInit THEN
	tonDelayDirectoryExist.IN := TRUE;
	//bError := TRUE;
	//sErrorString := F_GetTranslatedTxtEx("Directory does not exist", eLanguage); 
END_IF
END_METHOD

METHOD M_StartWrite : BOOL
VAR_INPUT
	saMessageTemp 		: ARRAY[0..iMaxIdxCsvData] OF WSTRING(255);
END_VAR
VAR
END_VAR

bStartWrite := TRUE;
saMessage := saMessageTemp;
END_METHOD

METHOD Reset : BOOL
VAR_INPUT
END_VAR
bError := FALSE;
sErrorString := "OK";

aWriteBuffer.bActive := FALSE;
bStartWrite := FALSE;
bInit := FALSE;
nStep := 0;
END_METHOD

METHOD Run
VAR_INPUT
END_VAR
tonDelayDirectoryExist(PT:=T#3S);

IF NOT Init() THEN
	RETURN;
END_IF

IF tonDelayDirectoryExist.Q AND NOT fbDirectory.bDirectoryExist THEN
	tonDelayDirectoryExist(IN:=FALSE);
	bError := TRUE;
	//sErrorString := F_GetTranslatedTxtEx("Directory does not exist", eLanguage); 
ELSIF tonDelayDirectoryExist.Q THEN
	tonDelayDirectoryExist(IN:=FALSE);
END_IF

IF sPath_OLD <> sPath THEN
	sPath_OLD := sPath;
	fbDirectory.Create(sPath);
	fbDirectory();
	IF NOT fbDirectory.bDirectoryExist THEN
		tonDelayDirectoryExist.IN := TRUE;
		//bError := TRUE;
		//sErrorString := F_GetTranslatedTxtEx("Directory does not exist", eLanguage); 
	END_IF
END_IF

WriteFile();
END_METHOD

METHOD PRIVATE WriteFile : BOOL

VAR
	///	logging text					
	
	ii		: INT;	
	nn		: INT;
END_VAR
(*	FILE LOG	*)
IF nStep = 0 THEN
	sFullPath := '';
	sFullPath := CONCAT(sPath, sDirSeparator);
	sFullPath := CONCAT(sFullPath, sYear);
	sFullPath := CONCAT(sFullPath, sMonth);
	sFullPath := CONCAT(sFullPath, sDay);
	sFullPath := CONCAT(sFullPath, '_');
	sFullPath := CONCAT(sFullPath, sFileName);
END_IF

CASE nStep OF

	0: 	// wait for write request
		hFile := 0; (*	empty File Handle	*)
		fbFileOpen(bExecute := FALSE);
		fbFileWrite(bExecute := FALSE);
		fbFileClose(bExecute := FALSE);
		fbEOF(bExecute := FALSE);
		fbFileRename(bExecute := FALSE);
		sText := '';
		IF bStartWrite AND bInit AND NOT bError THEN
			bStartWrite := FALSE;
			aWriteBuffer.bActive := TRUE;
			nStep := 10;	
		END_IF		

	10: (*	open file	*)
		fbFileOpen(sPathName := sFullPath,
					nMode := FOPEN_MODEAPPEND OR FOPEN_MODEPLUS,
					ePath := PATH_GENERIC,
					bExecute := TRUE,
					tTimeout := T#2S,
					hFile => hFile);
		IF NOT fbFileOpen.bBusy THEN
			IF NOT fbFileOpen.bError THEN
				fbFileOpen(bExecute := FALSE);			
				nStep := 20;
			ELSE				
				nStep := 1000; (*	error	*)
				bError := TRUE;
				//sErrorString := F_GetTranslatedTxtEx("Open File failed", eLanguage); 
			END_IF
		END_IF
		
	20: (* get next log item *)
		stOrderData REF= 0;

		IF aWriteBuffer.bActive THEN
			stOrderData REF= aWriteBuffer;
		END_IF
		
		IF __ISVALIDREF(stOrderData) THEN // found
			nStep := 30;
		ELSE
			nStep := 50; // not found - ready
			//bError := TRUE;
			//sErrorString := 'no reference found';
		END_IF

	30: (*	check end of file (max size)	*)
		fbEOF(hFile := hFile,
			bExecute := TRUE,
			tTimeout := T#2S);
		IF NOT fbEOF.bBusy THEN
			IF NOT fbEOF.bError THEN
				fbEOF(bExecute:= FALSE);				
				IF NOT fbEOF.bEOF THEN
					iMessageCount:=0;
					nStep := 40;
				ELSE					
					nStep := 100;
				END_IF
			ELSE				
				nStep := 0; (*	error	*)
				bError := TRUE;
				//sErrorString := F_GetTranslatedTxtEx("error: end of file", eLanguage);
			END_IF
		END_IF	
		
	40:
		sText:=WSTRING_TO_STRING(saMessage[iMessageCount]);	
		sText := CONCAT(sText, ';');
		//sText := CONCAT(sText, '$R');
		
		nStep := 45;
		
	45: (*	write Data 1/2	*)
		//sText:="";
		//FOR nn:=0 TO (iMaxCSVdata(*/2*)) BY 1 DO
		//	sText := WCONCAT(sText, saMessage[nn]);
		//	sText := WCONCAT(sText, ";");
		//END_FOR
		///sText := CONCAT(sText, '$R');

		fbFileWrite(hFile := hFile,
					pWriteBuff := ADR(sText),
					cbWriteLen := INT_TO_UINT(LEN(sText)),
					bExecute := TRUE,
					tTimeout := T#2S);
		IF NOT fbFileWrite.bBusy THEN
			IF NOT fbFileWrite.bError THEN
				stOrderData.bActive := FALSE;
				fbFileWrite(bExecute := FALSE);	
				sText := '';		
				fbFileWrite(pWriteBuff := ADR(sText));
				//nStep := 45;
				IF (iMessageCount < iMaxIdxCsvData) AND (saMessage[iMessageCount]<>"") THEN
					iMessageCount:=iMessageCount+1;
					nStep := 40;
				ELSE
					iMessageCount:=0;
					nStep := 46;
				END_IF		
			ELSE				
				nStep := 0; (*	error	*)
			END_IF
		END_IF


	46: (*	write Data 1/2	*)
		sText :='$N';

		fbFileWrite(hFile := hFile,
					pWriteBuff := ADR(sText),
					cbWriteLen := INT_TO_UINT(LEN(sText)),
					bExecute := TRUE,
					tTimeout := T#2S);
		IF NOT fbFileWrite.bBusy THEN
			IF NOT fbFileWrite.bError THEN
				stOrderData.bActive := FALSE;
				fbFileWrite(bExecute := FALSE);	
				sText := '';		
				fbFileWrite(pWriteBuff := ADR(sText));
				nStep := 20;	
			ELSE				
				nStep := 0; (*	error	*)
			END_IF
		END_IF




		
//	45:(*	write Data 2/2	*)
//		FOR nn:=((iMaxCSVdata/2)+1) TO iMaxCSVdata BY 1 DO
//			sText := WCONCAT(sText, saMessage[nn]);
//			sText := WCONCAT(sText, ";");
//		END_FOR
//		sText := WCONCAT(sText, "$R");
//		
//		fbFileWrite(hFile := hFile,
//					pWriteBuff := ADR(sText),
//					cbWriteLen := INT_TO_UINT(WLEN(sText)),
//					bExecute := TRUE,
//					tTimeout := T#2S);
//		IF NOT fbFileWrite.bBusy THEN
//			IF NOT fbFileWrite.bError THEN
//				stOrderData.bActive := FALSE;
//				fbFileWrite(bExecute := FALSE);				
//				nStep := 20;
//			ELSE				
//				nStep := 0; (*	error	*)
//			END_IF
//		END_IF

	50: (*	File Close	*)
		fbFileClose(hFile := hFile,
				bExecute := TRUE,
				tTimeout := T#2S);
		IF NOT fbFileClose.bBusy THEN
			IF NOT fbFileClose.bError THEN
				nStep := 60; (*	done	*)
			ELSE
				nStep := 0; (*	error	*)
			END_IF
		END_IF
		
	60:	// run delay
		tonDelay(IN := TRUE, PT := tWriteFilter);
		IF tonDelay.Q THEN
			tonDelay(IN := FALSE);
			nStep := 0;
		END_IF
		
	100: (*	close file for rename	*)
		fbFileClose(hFile := hFile,
					bExecute := TRUE,
					tTimeout := T#2S);
		IF NOT fbFileClose.bBusy THEN
			IF NOT fbFileClose.bError THEN
				fbFileClose(bExecute := FALSE);
				nStep := 110;
			ELSE
				nStep := 0;
			END_IF
		END_IF

	110: (*	Rename full file	*)
		sPathNew := '';
		sPathNew := CONCAT(sPath, sDirSeparator);
		
		sPathNew := CONCAT(sPathNew, sTimeString);
		sPathNew := CONCAT(sPathNew,'.log');
		
		fbFileRename(sOldName := sFullPath,
					sNewName := sPathNew ,
					ePath := PATH_GENERIC ,
					bExecute := TRUE ,
					tTimeout := T#2S);
		IF NOT fbFileRename.bBusy THEN
			IF NOT fbFileRename.bError THEN
				nStep := 10; (*	new try	*)
			ELSE
				nStep := 0;
			END_IF
		END_IF
END_CASE
END_METHOD

END_FUNCTION_BLOCK

// ---- POUs/System/Utilities/FB_JogTrigTon.TcPOU
FUNCTION_BLOCK FB_JogTrigTon
VAR_INPUT
	// jog +
	bJogP : BOOL;
	// jog -
	bJogN : BOOL;
	// ton time
	tTime : TIME := T#1S;	
END_VAR
VAR_OUTPUT
	// jog + falling flag
	fQp : BOOL;
	// jog - falling flag
	fQn : BOOL;
	// jog +/- timer flag
	tQ : BOOL;
	// jog +/- or flag
	bOr : BOOL;
	// jog + timer flag
	bTmrJogP : BOOL;
	// jog - timer flag
	bTmrJogN : BOOL;
END_VAR
VAR
	ftrigP	: F_TRIG;
	ftrigN	: F_TRIG;
	tonTm	: TON;
	btQ		: BOOL;
END_VAR

bOr := bJogP OR bJogN;
ftrigP(CLK := bJogP, Q => fQp);
ftrigN(CLK := bJogN, Q => fQn);
tonTm(IN := bOr, PT := tTime, Q => tQ);
bTmrJogP := bJogP AND tQ;
bTmrJogN := bJogN AND tQ;

IF tQ THEN
	btQ := TRUE;
ELSIF btQ AND (fQp OR fQn) THEN
	btQ := FALSE;
END_IF

END_FUNCTION_BLOCK

// ---- POUs/System/Utilities/FB_Puls_On_Off.TcPOU
FUNCTION_BLOCK FB_Puls_On_Off
VAR_INPUT
	bEnable		: BOOL;
	tPulsOn		: TIME:= T#5S;
	tPulsOff	: TIME:= T#5S;
END_VAR
VAR_OUTPUT
	bOut		: BOOL;
END_VAR
VAR
	tonPulsOn	: ton;
	tonPulsOff	: ton;	
END_VAR


tonPulsOn.PT:=tPulsOn;
tonPulsOn();
tonPulsOn.IN:=NOT tonPulsOff.Q AND bEnable;

tonPulsOff.PT:=tPulsOff;
tonPulsOff();
tonPulsOff.IN:=tonPulsOn.Q;

bOut:=NOT tonPulsOn.Q AND bEnable;

END_FUNCTION_BLOCK

// ---- POUs/System/Utilities/FB_RtrigFtrigTof.TcPOU
FUNCTION_BLOCK PUBLIC FB_RtrigFtrigTof
VAR_INPUT
	bIn : BOOL;
	tPt : TIME := T#0S;
END_VAR
VAR_OUTPUT
	// rising trigger bIn
	bRq : BOOL;
	// falling trigger after tPt
	bFq : BOOL;
END_VAR
VAR
	fbTof : TOF;
	rtrig : R_TRIG;
	ftrig : F_TRIG;
END_VAR

fbTof(IN:= bIn, PT := tPt);
rtrig(CLK := fbTof.Q, Q => bRq);
ftrig(CLK := fbTof.Q, Q => bFq);

END_FUNCTION_BLOCK

// ---- POUs/System/Utilities/FB_StableValue.TcPOU
FUNCTION_BLOCK FB_StableValue //stabiler wert
VAR_INPUT
	fValue		: LREAL;
	iPrecision	: INT;
	bRound		: BOOL;
	tStabileTon	: TIME := T#50MS;
	tStabileTof	: TIME := T#20MS;
END_VAR
VAR_OUTPUT
	sValue				: STRING;
	fValueFmt			: LREAL;
	bStabileValue		: BOOL;
	bStabileValueTout	: BOOL;
END_VAR
VAR
	fTempValue	: LREAL;
	tonStabile	: TON;
	tofStabile	: TOf;
END_VAR


sValue := LREAL_TO_FMTSTR(fValue,iPrecision,bRound);
fValueFmt := TO_LREAL(sValue);

IF (fValueFmt <> fTempValue) THEN
	fTempValue := fValueFmt;
END_IF
bStabileValue := (fValueFmt = fTempValue);

tonStabile.IN := bStabileValue;
tonStabile.PT := tStabileTon;
tonStabile();

tofStabile.IN := tonStabile.Q;
tofStabile.PT := tStabileTof;
tofStabile();

bStabileValueTout := tofStabile.Q;

END_FUNCTION_BLOCK

// ---- POUs/System/Utilities/FB_ToggleSwitch.TcPOU
FUNCTION_BLOCK FB_ToggleSwitch
VAR_INPUT
	EN		:BOOL;			(*FB enable*)
	IN		:BOOL;			(*if IN is true then FC_CurrentimputSwitch = true -> if IN is already true then FC_CurrentimputSwitch = false*)
	RESET	:BOOL;			(* if RESET is  true then FC_CurrentimputSwitch = false*)
END_VAR
VAR_OUTPUT
	ACT		:BOOL;
	OUT		:BOOL;
	INVOUT	:BOOL;
END_VAR
VAR_IN_OUT
	INOUT	:BOOL;
END_VAR
VAR
	HM		:BOOL;
END_VAR

(*	Version history:	FB toggle switch

	DATE	|	Version	|	TwinCAT		|	PLC Control Version	|		Author				|		Comments
----------------------------------------------------------------------------------------------------------------------------------------------------------------------------------------------------------------
 2011-06-18	|	1.0		|	v2.11.xxx		|	v2.11.0 (Build 1804)	| www.rmth.at/Günther Müllner	| Orig. program for RMTH
***********************************************************************************************************************************************************************)
IF EN THEN
	ACT:=IN;
	IF IN AND NOT HM THEN
		INOUT:=TRUE;
	END_IF
	IF NOT IN AND INOUT THEN
		HM:=TRUE;
	END_IF
	IF (IN AND INOUT AND HM) OR RESET THEN
		INOUT:=FALSE;
	END_IF
	IF NOT IN AND NOT INOUT THEN
		HM:=FALSE;
	END_IF
	OUT:=INOUT;
	INVOUT	:= NOT INOUT;
ELSE
	INOUT:=FALSE;
	OUT:=FALSE;
	INVOUT:=FALSE;
END_IF

END_FUNCTION_BLOCK

// ---- POUs/System/Utilities/Functions/F_ADD_REF_F.TcPOU
FUNCTION F_ADD_REF_F : BOOL
VAR_IN_OUT
	fValueRoot	: LREAL;
END_VAR
VAR_INPUT
	fValue		: LREAL;
END_VAR

fValueRoot := fValueRoot + fValue;

END_FUNCTION

// ---- POUs/System/Utilities/Functions/F_Byte_To_DWord.TcPOU
FUNCTION F_Byte_To_DWord : DWORD
VAR_INPUT
	bByte0	: BYTE;
	bByte1	: BYTE;
	bByte2	: BYTE;
	bByte3	: BYTE;
END_VAR
VAR
END_VAR

MEMCPY(ADR(F_Byte_To_DWord),ADR(bByte0),SIZEOF(bByte0)); (*set  zero*)
MEMCPY(ADR(F_Byte_To_DWord)+1,ADR(bByte1),SIZEOF(bByte0)); (*set  zero*)
MEMCPY(ADR(F_Byte_To_DWord)+2,ADR(bByte2),SIZEOF(bByte0)); (*set  zero*)
MEMCPY(ADR(F_Byte_To_DWord)+3,ADR(bByte3),SIZEOF(bByte0)); (*set  zero*)

END_FUNCTION

// ---- POUs/System/Utilities/Functions/F_Byte_To_Word.TcPOU
FUNCTION F_Byte_To_Word : WORD
VAR_INPUT
	bByte0	: BYTE;
	bByte1	: BYTE;
END_VAR
VAR
END_VAR

MEMCPY(ADR(F_Byte_To_Word),ADR(bByte0),SIZEOF(bByte0)); (*set  zero*)
MEMCPY(ADR(F_Byte_To_Word)+1,ADR(bByte1),SIZEOF(bByte0)); (*set  zero*)

END_FUNCTION

// ---- POUs/System/Utilities/Functions/F_FormatString.TcPOU
FUNCTION F_FormatString : String
VAR_INPUT
	sInput,
	sPrefix		:STRING;
	nLenght		:INT;
END_VAR
VAR
	nPosition	:INT;
END_VAR

nPosition := FIND(sInput,sPrefix);
F_FormatString := LEFT(sInput,(nPosition + nLenght));

END_FUNCTION

// ---- POUs/System/Utilities/Functions/F_InRange.TcPOU
FUNCTION F_InRange : BOOL
VAR_INPUT
	fValue			: LREAL;	//11.5
	fLowerLimit		: LREAL;	//10
	fUpperLimit		: LREAL;	//12	
END_VAR
VAR
	fTempUl			: LREAL;
	fTempLl			: LREAL;
END_VAR

F_InRange:=(fValue >= fLowerLimit) AND (fValue <= fUpperLimit);

END_FUNCTION

// ---- POUs/System/Utilities/Functions/F_Log_Add.TcPOU
FUNCTION F_Log_Add : STRING
VAR_INPUT
	sString		: STRING;
END_VAR
VAR_IN_OUT
	sTemp		: STRING;
	sLog1_100	: ARRAY[0..100] OF STRING;
END_VAR
VAR
	ii 			: INT;
END_VAR

IF sTemp = sString THEN
	RETURN;
END_IF

FOR ii := 0 TO 99 DO
	sLog1_100[ii + 1] := sLog1_100[ii];
END_FOR

sLog1_100[0] := sString;
sTemp := sString;

END_FUNCTION

// ---- POUs/System/Utilities/Functions/F_Real_To_Byte.TcPOU
FUNCTION F_Real_To_Byte : BYTE
VAR_INPUT
	nByte	: INT; //x (1 - 4) byte it get from real
	fReal	: REAL;	 
END_VAR
VAR
	nPos	: LWORD;
END_VAR


CASE nByte OF
	1:
		nPos := 0;
	2:
		nPos := 7;
	3:
		nPos := 14;
	4:
		nPos := 21;
ELSE
	RETURN;	
END_CASE

MEMCPY(ADR(F_Real_To_Byte),(ADR(fReal)+ nPos),8);

END_FUNCTION

// ---- POUs/System/Utilities/Functions/F_Settings_Row_Delete.TcPOU
FUNCTION F_Settings_Row_Delete : BOOL
VAR_IN_OUT
	aSettings	: ARRAY[*] OF ST_Data_Item; /// settings structure
END_VAR
VAR_INPUT
	nPlace				:INT;
END_VAR
VAR
	nn	: DINT;
END_VAR

IF (nPlace < LOWER_BOUND(aSettings,1)) OR (nPlace > UPPER_BOUND(aSettings,1)) THEN
	RETURN;
END_IF

//Check Array Size
MEMSET(ADR(aSettings[nPlace]),0,SIZEOF(aSettings[nPlace])); (*set  zero*)

FOR nn:= nPlace TO UPPER_BOUND(aSettings,1) BY 1 DO
	MEMCPY(ADR(aSettings[nn]),ADR(aSettings[nn+1]),SIZEOF(aSettings[nn+1]));		
END_FOR
//delete last row
MEMSET(ADR(aSettings[UPPER_BOUND(aSettings,1)]),0,SIZEOF(aSettings[UPPER_BOUND(aSettings,1)])); (*set  zero*)

END_FUNCTION

// ---- POUs/System/Utilities/Functions/F_Settings_Row_Insert.TcPOU
FUNCTION F_Settings_Row_Insert : BOOL
VAR_IN_OUT
	aSettings	: ARRAY[*] OF ST_Data_Item; /// settings structure
END_VAR
VAR_INPUT
	nPlace				:INT;
	//stGroup				:ST_Text;
	//stName				:ST_Text;
	//stUnit				:ST_Text;
	//eDataType			:E_DataType;
END_VAR
VAR
	nn	: DINT;
END_VAR

IF (nPlace < LOWER_BOUND(aSettings,1)) OR (nPlace > UPPER_BOUND(aSettings,1)) THEN
	RETURN;
END_IF

//Check Array Size

FOR nn:= (UPPER_BOUND(aSettings,1)-1) TO  MAX(LOWER_BOUND(aSettings,1),nPlace) by -1 DO
	MEMCPY(ADR(aSettings[nn+1]),ADR(aSettings[nn]),SIZEOF(aSettings[nn+1])); (*set  zero*)		
END_FOR
MEMSET(ADR(aSettings[nPlace]),0,SIZEOF(aSettings[nPlace])); (*set  zero*)

END_FUNCTION

// ---- POUs/System/Utilities/Functions/F_Trend.TcPOU
FUNCTION F_Trend : BOOL
VAR_INPUT
	fCurrentValue	: REAL;
END_VAR
VAR_IN_OUT
	fValueMax		: REAL;
	fValueMin		: REAL;	
END_VAR

IF (fCurrentValue > fValueMax) THEN
	fValueMax:=fCurrentValue;
ELSIF (fCurrentValue < fValueMax) THEN
	fValueMin:= fCurrentValue;
END_IF

END_FUNCTION

// ---- POUs/System/Utilities/String/WConcat10.TcPOU
FUNCTION WConcat10 : WSTRING(255)
VAR_INPUT
	wsExpression1: WSTRING(255);
	wsExpression2: WSTRING(255);
	wsExpression3: WSTRING(255);
	wsExpression4: WSTRING(255);
	wsExpression5: WSTRING(255);
	wsExpression6: WSTRING(255);
	wsExpression7: WSTRING(255);
	wsExpression8: WSTRING(255);
	wsExpression9: WSTRING(255);
	wsExpression10: WSTRING(255);
END_VAR

WConcat10 := WCONCAT(wsExpression1, wsExpression2);
WConcat10 := WCONCAT(WConcat10, wsExpression3);
WConcat10 := WCONCAT(WConcat10, wsExpression4);
WConcat10 := WCONCAT(WConcat10, wsExpression5);
WConcat10 := WCONCAT(WConcat10, wsExpression6);
WConcat10 := WCONCAT(WConcat10, wsExpression7);
WConcat10 := WCONCAT(WConcat10, wsExpression8);
WConcat10 := WCONCAT(WConcat10, wsExpression9);
WConcat10 := WCONCAT(WConcat10, wsExpression10);

END_FUNCTION

// ---- POUs/System/Utilities/String/WConcat4.TcPOU
FUNCTION WConcat4 : WSTRING(255)
VAR_INPUT
	wsExpression1: WSTRING(255);
	wsExpression2: WSTRING(255);
	wsExpression3: WSTRING(255);
	wsExpression4: WSTRING(255);
END_VAR

WConcat4 := WCONCAT(wsExpression1, wsExpression2);
WConcat4 := WCONCAT(WConcat4, wsExpression3);
WConcat4 := WCONCAT(WConcat4, wsExpression4);

END_FUNCTION

// ---- POUs/System/Utilities/String/WConcat5.TcPOU
FUNCTION WConcat5 : WSTRING(255)
VAR_INPUT
	wsExpression1: WSTRING(255);
	wsExpression2: WSTRING(255);
	wsExpression3: WSTRING(255);
	wsExpression4: WSTRING(255);
	wsExpression5: WSTRING(255);
END_VAR

WConcat5 := WCONCAT(wsExpression1, wsExpression2);
WConcat5 := WCONCAT(WConcat5, wsExpression3);
WConcat5 := WCONCAT(WConcat5, wsExpression4);
WConcat5 := WCONCAT(WConcat5, wsExpression5);

END_FUNCTION

// ---- POUs/System/Utilities/String/WConcat6.TcPOU
FUNCTION WConcat6 : WSTRING(255)
VAR_INPUT
	wsExpression1: WSTRING(255);
	wsExpression2: WSTRING(255);
	wsExpression3: WSTRING(255);
	wsExpression4: WSTRING(255);
	wsExpression5: WSTRING(255);
	wsExpression6: WSTRING(255);
END_VAR

WConcat6 := WCONCAT(wsExpression1, wsExpression2);
WConcat6 := WCONCAT(WConcat6, wsExpression3);
WConcat6 := WCONCAT(WConcat6, wsExpression4);
WConcat6 := WCONCAT(WConcat6, wsExpression5);
WConcat6 := WCONCAT(WConcat6, wsExpression6);

END_FUNCTION

// ---- POUs/System/Utilities/String/WConcat7.TcPOU
FUNCTION WConcat7 : WSTRING(255)
VAR_INPUT
	wsExpression1: WSTRING(255);
	wsExpression2: WSTRING(255);
	wsExpression3: WSTRING(255);
	wsExpression4: WSTRING(255);
	wsExpression5: WSTRING(255);
	wsExpression6: WSTRING(255);
	wsExpression7: WSTRING(255);
END_VAR

WConcat7 := WCONCAT(wsExpression1, wsExpression2);
WConcat7 := WCONCAT(WConcat7, wsExpression3);
WConcat7 := WCONCAT(WConcat7, wsExpression4);
WConcat7 := WCONCAT(WConcat7, wsExpression5);
WConcat7 := WCONCAT(WConcat7, wsExpression6);
WConcat7 := WCONCAT(WConcat7, wsExpression7);

END_FUNCTION

// ---- POUs/System/Utilities/String/WConcat8.TcPOU
FUNCTION WConcat8 : WSTRING(255)
VAR_INPUT
	wsExpression1: WSTRING(255);
	wsExpression2: WSTRING(255);
	wsExpression3: WSTRING(255);
	wsExpression4: WSTRING(255);
	wsExpression5: WSTRING(255);
	wsExpression6: WSTRING(255);
	wsExpression7: WSTRING(255);
	wsExpression8: WSTRING(255);
END_VAR

WConcat8 := WCONCAT(wsExpression1, wsExpression2);
WConcat8 := WCONCAT(WConcat8, wsExpression3);
WConcat8 := WCONCAT(WConcat8, wsExpression4);
WConcat8 := WCONCAT(WConcat8, wsExpression5);
WConcat8 := WCONCAT(WConcat8, wsExpression6);
WConcat8 := WCONCAT(WConcat8, wsExpression7);
WConcat8 := WCONCAT(WConcat8, wsExpression8);

END_FUNCTION

// ---- POUs/System/Utilities/String/WConcat9.TcPOU
FUNCTION WConcat9 : WSTRING(255)
VAR_INPUT
	wsExpression1: WSTRING(255);
	wsExpression2: WSTRING(255);
	wsExpression3: WSTRING(255);
	wsExpression4: WSTRING(255);
	wsExpression5: WSTRING(255);
	wsExpression6: WSTRING(255);
	wsExpression7: WSTRING(255);
	wsExpression8: WSTRING(255);
	wsExpression9: WSTRING(255);
END_VAR

WConcat9 := WCONCAT(wsExpression1, wsExpression2);
WConcat9 := WCONCAT(WConcat9, wsExpression3);
WConcat9 := WCONCAT(WConcat9, wsExpression4);
WConcat9 := WCONCAT(WConcat9, wsExpression5);
WConcat9 := WCONCAT(WConcat9, wsExpression6);
WConcat9 := WCONCAT(WConcat9, wsExpression7);
WConcat9 := WCONCAT(WConcat9, wsExpression8);
WConcat9 := WCONCAT(WConcat9, wsExpression9);

END_FUNCTION
